(* Logix 5000 project; controller fun_probably 1769-L16ER-BB1B rev 34.12; software revision 34.01 *)

TASK MainTask (continuous, watchdog 500 ms) : MainProgram

MODULES
   Local : 1769-L16ER-BB1B (PointIO 0, rev 34.12)
      Discrete_IO : Embedded (PointIO 1, rev 34.11, Output RPI 20 ms)
           Local:1:I.Data.3   // Main or Troubleshooting Switch
END_MODULES

VAR_GLOBAL   (* controller tags *)
   bestScore : DINT;
   birdDownHit : REAL;
   birdFrontHit : REAL[2];
   birdUpHit : REAL;
   birdXPos : DINT;
   birdYPos : REAL;
   clock : TIMER := (PRE := 50);
   downSpeed : DINT;
   dX : DINT;
   dY : REAL;
   fallFunctionX : COUNTER := (PRE := 10);
   fastestFall : BOOL;
   getOffset1 : BOOL;
   getOffset2 : BOOL;
   GodMode : BOOL;
   gravity : REAL;
   halt : BOOL;
   HMI_Start : BOOL;
   increment : DINT;
   intermediateVal : REAL;
   invertUpSpeed : DINT;
   limit : DINT;
   loseBit : BOOL;
   multiplier : DINT;
   offset : DINT;
   ons1 : BOOL;
   ons10 : BOOL;
   ons11 : BOOL;
   ons12 : BOOL;
   ons13 : BOOL;
   ons14 : BOOL;
   ons15 : BOOL;
   ons16 : BOOL;
   ons2 : BOOL;
   ons3 : BOOL;
   ons4 : BOOL;
   ons5 : BOOL;
   ons6 : BOOL;
   ons7 : BOOL;
   ons8 : BOOL;
   ons9 : BOOL;
   pipe1_collision : BOOL;
   pipe1_reset : BOOL;
   pipe1XPos : DINT;
   pipe1Y : REAL;
   pipe1Ybot : REAL;
   pipe1Yhit : DINT;
   pipe2_collision : BOOL;
   pipe2_reset : BOOL;
   pipe2XPos : DINT;
   pipe2Y : DINT;
   pipe2Ybot : DINT;
   pipe2Yhit : DINT;
   run_pipe2 : BOOL;
   score : COUNTER;
   seed : DINT;
   speed : DINT;
   startCR : BOOL;
   temp_offset : DINT;
   temp_seed : DINT;
   test : REAL[32];
   upSpeed : DINT;
END_VAR

PROGRAM MainProgram   (* main routine MainRoutine *)

ROUTINE MainRoutine   (* ladder *)
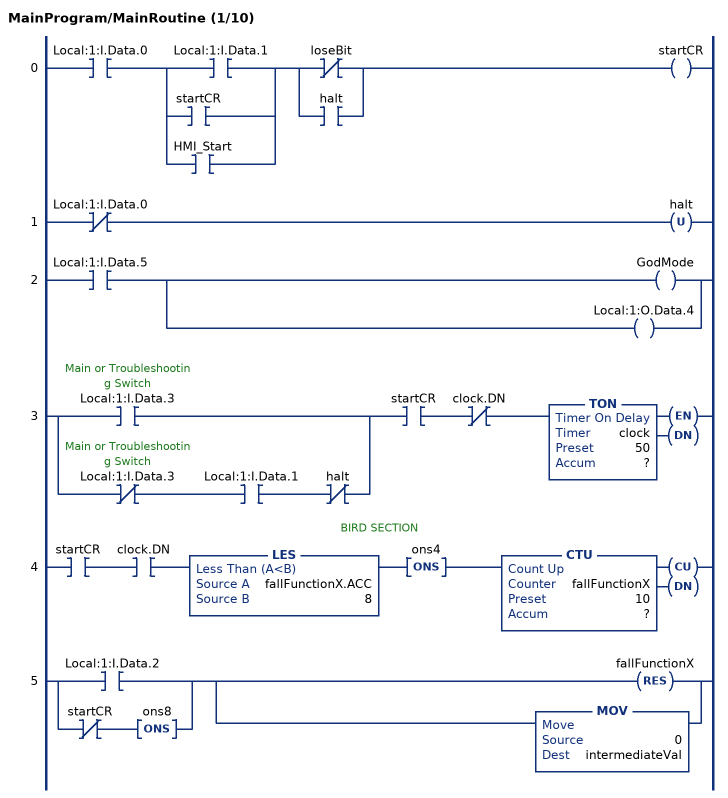
   0: XIC(Local:1:I.Data.0)[XIC(Local:1:I.Data.1) ,[XIC(startCR) ,XIC(HMI_Start) ] ][XIO(loseBit) ,XIC(halt) ]OTE(startCR);
   1: XIO(Local:1:I.Data.0)OTU(halt);
   2: XIC(Local:1:I.Data.5)[OTE(GodMode) ,OTE(Local:1:O.Data.4) ];
   3: [XIC(Local:1:I.Data.3) ,XIO(Local:1:I.Data.3) XIC(Local:1:I.Data.1) XIO(halt) ]XIC(startCR)XIO(clock.DN)TON(clock,?,?);
   // BIRD SECTION
   4: XIC(startCR)XIC(clock.DN)LES(fallFunctionX.ACC,8)ONS(ons4)CTU(fallFunctionX,?,?);
   5: [XIC(Local:1:I.Data.2) ,XIO(startCR) ONS(ons8) ][RES(fallFunctionX) ,MOV(0,intermediateVal) ];
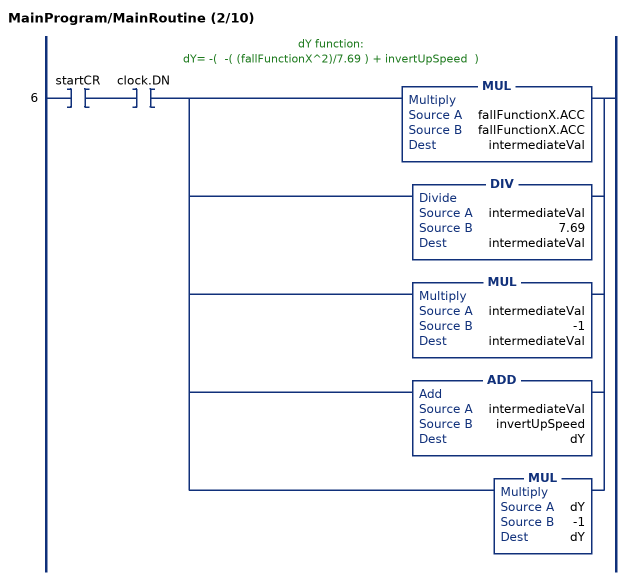
   // dY function:
   // dY= -(  -( (fallFunctionX^2)/7.69 ) + invertUpSpeed  )
   6: XIC(startCR)XIC(clock.DN)[MUL(fallFunctionX.ACC,fallFunctionX.ACC,intermediateVal) ,[DIV(intermediateVal,7.69,intermediateVal) ,[MUL(intermediateVal,-1,intermediateVal) ,[ADD(intermediateVal,invertUpSpeed,dY) ,MUL(dY,-1,dY) ] ] ] ];
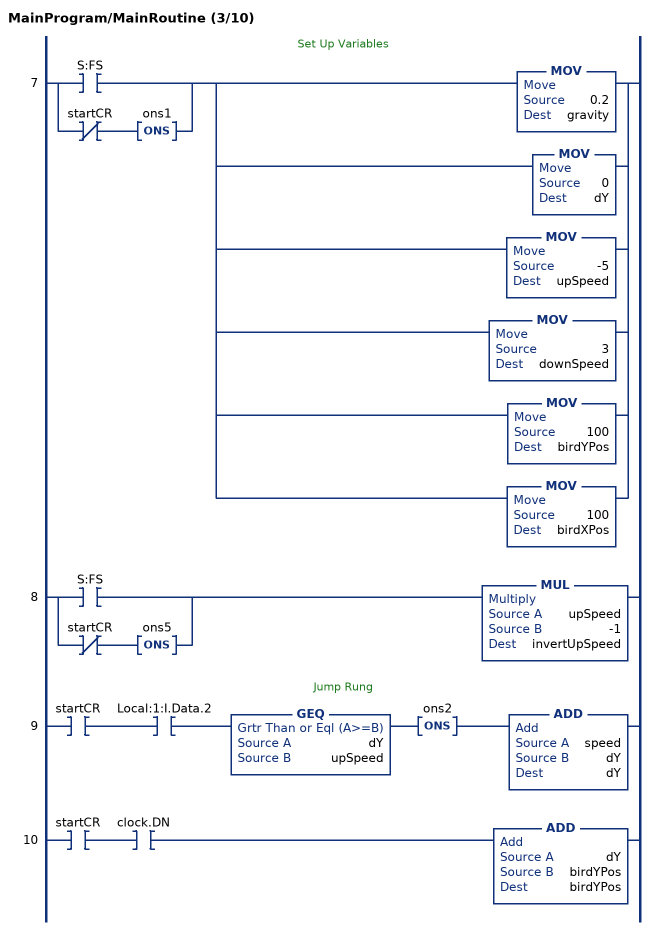
   // Set Up Variables
   7: [XIC(S:FS) ,XIO(startCR) ONS(ons1) ][MOV(0.2,gravity) ,[MOV(0,dY) ,[MOV(-5,upSpeed) ,[MOV(3,downSpeed) ,[MOV(100,birdYPos) ,MOV(100,birdXPos) ] ] ] ] ];
   8: [XIC(S:FS) ,XIO(startCR) ONS(ons5) ]MUL(upSpeed,-1,invertUpSpeed);
   // Jump Rung
   9: XIC(startCR)XIC(Local:1:I.Data.2)GEQ(dY,upSpeed)ONS(ons2)ADD(speed,dY,dY);
   10: XIC(startCR)XIC(clock.DN)ADD(dY,birdYPos,birdYPos);
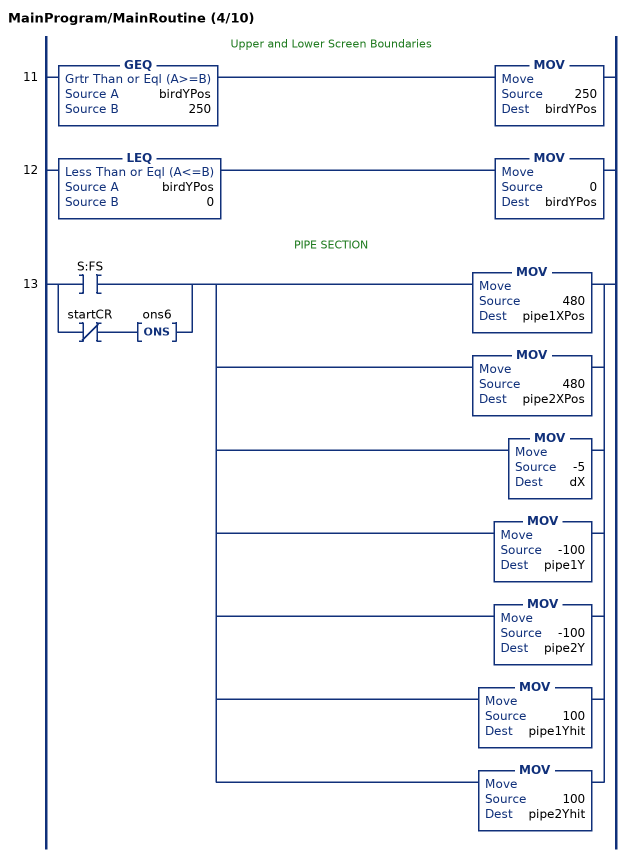
   // Upper and Lower Screen Boundaries
   11: GEQ(birdYPos,250)MOV(250,birdYPos);
   12: LEQ(birdYPos,0)MOV(0,birdYPos);
   // PIPE SECTION
   13: [XIC(S:FS) ,XIO(startCR) ONS(ons6) ][[MOV(480,pipe1XPos) ,MOV(480,pipe2XPos) ] ,[MOV(-5,dX) ,[[MOV(-100,pipe1Y) ,MOV(-100,pipe2Y) ] ,[MOV(100,pipe1Yhit) ,MOV(100,pipe2Yhit) ] ] ] ];
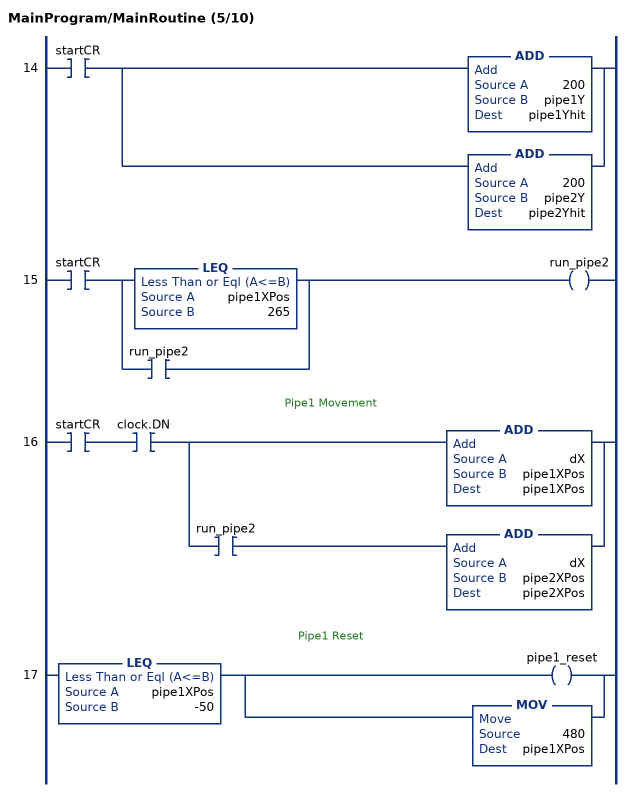
   14: XIC(startCR)[ADD(200,pipe1Y,pipe1Yhit) ,ADD(200,pipe2Y,pipe2Yhit) ];
   15: XIC(startCR)[LEQ(pipe1XPos,265) ,XIC(run_pipe2) ]OTE(run_pipe2);
   // Pipe1 Movement
   16: XIC(startCR)XIC(clock.DN)[ADD(dX,pipe1XPos,pipe1XPos) ,XIC(run_pipe2) ADD(dX,pipe2XPos,pipe2XPos) ];
   // Pipe1 Reset
   17: LEQ(pipe1XPos,-50)[OTE(pipe1_reset) ,MOV(480,pipe1XPos) ];
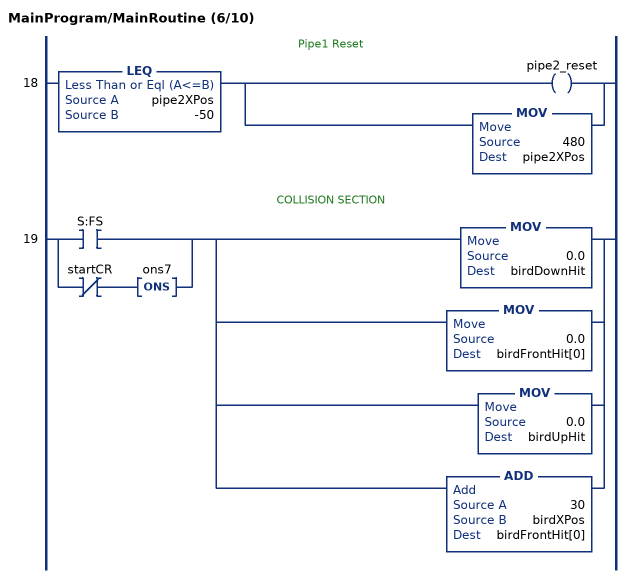
   // Pipe1 Reset
   18: LEQ(pipe2XPos,-50)[OTE(pipe2_reset) ,MOV(480,pipe2XPos) ];
   // COLLISION SECTION
   19: [XIC(S:FS) ,XIO(startCR) ONS(ons7) ][MOV(0.0,birdDownHit) ,[MOV(0.0,birdFrontHit[0]) ,[MOV(0.0,birdUpHit) ,ADD(30,birdXPos,birdFrontHit[0]) ] ] ];
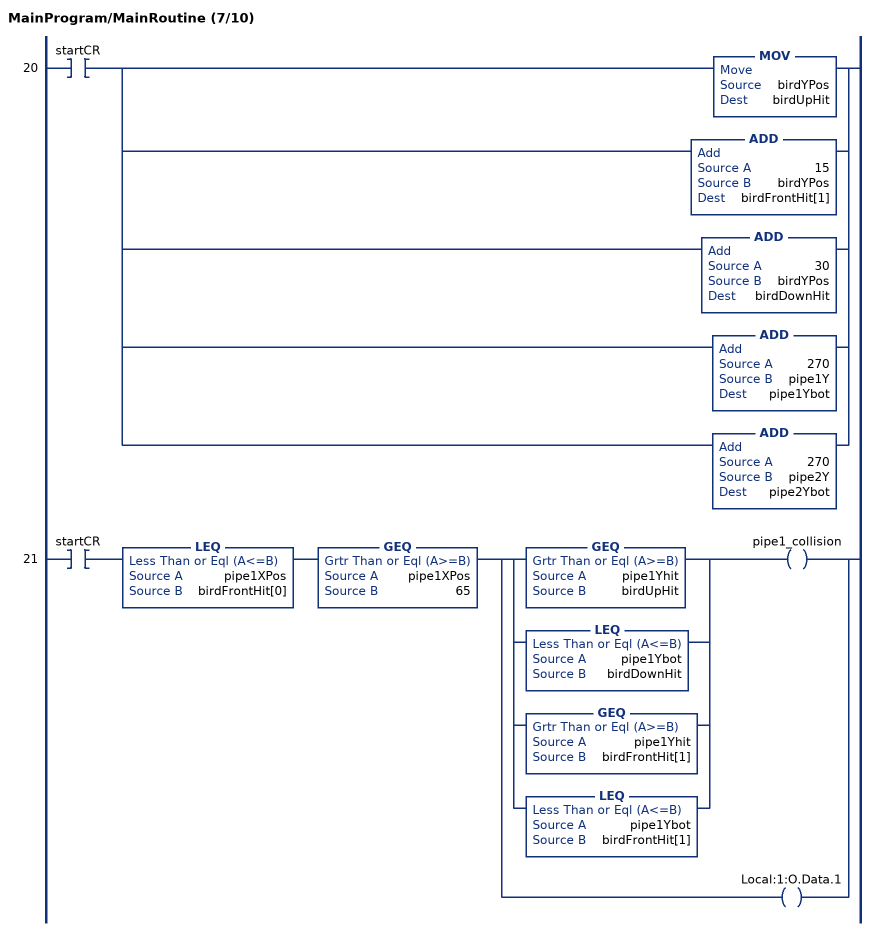
   20: XIC(startCR)[MOV(birdYPos,birdUpHit) ,[ADD(15,birdYPos,birdFrontHit[1]) ,[ADD(30,birdYPos,birdDownHit) ,[ADD(270,pipe1Y,pipe1Ybot) ,ADD(270,pipe2Y,pipe2Ybot) ] ] ] ];
   21: XIC(startCR)LEQ(pipe1XPos,birdFrontHit[0])GEQ(pipe1XPos,65)[[[GEQ(pipe1Yhit,birdUpHit) ,LEQ(pipe1Ybot,birdDownHit) ] ,[GEQ(pipe1Yhit,birdFrontHit[1]) ,LEQ(pipe1Ybot,birdFrontHit[1]) ] ] OTE(pipe1_collision) ,OTE(Local:1:O.Data.1) ];
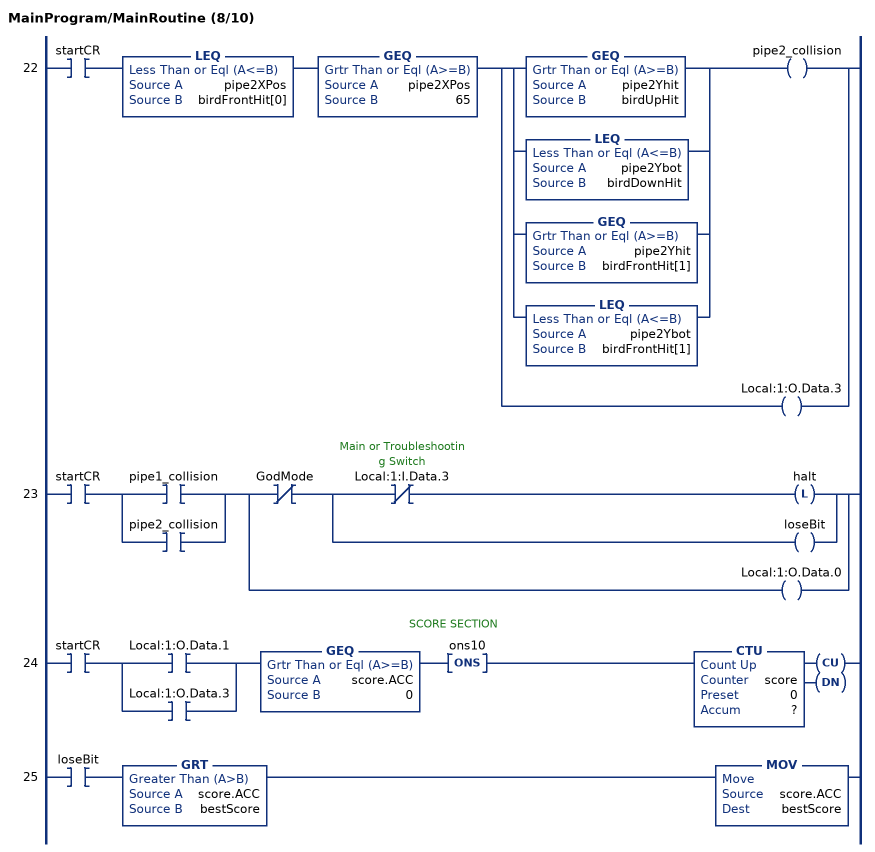
   22: XIC(startCR)LEQ(pipe2XPos,birdFrontHit[0])GEQ(pipe2XPos,65)[[[GEQ(pipe2Yhit,birdUpHit) ,LEQ(pipe2Ybot,birdDownHit) ] ,[GEQ(pipe2Yhit,birdFrontHit[1]) ,LEQ(pipe2Ybot,birdFrontHit[1]) ] ] OTE(pipe2_collision) ,OTE(Local:1:O.Data.3) ];
   23: XIC(startCR)[XIC(pipe1_collision) ,XIC(pipe2_collision) ][XIO(GodMode) [XIO(Local:1:I.Data.3) OTL(halt) ,OTE(loseBit) ] ,OTE(Local:1:O.Data.0) ];
   // SCORE SECTION
   24: XIC(startCR)[XIC(Local:1:O.Data.1) ,XIC(Local:1:O.Data.3) ]GEQ(score.ACC,0)ONS(ons10)CTU(score,?,?);
   25: XIC(loseBit)GRT(score.ACC,bestScore)MOV(score.ACC,bestScore);
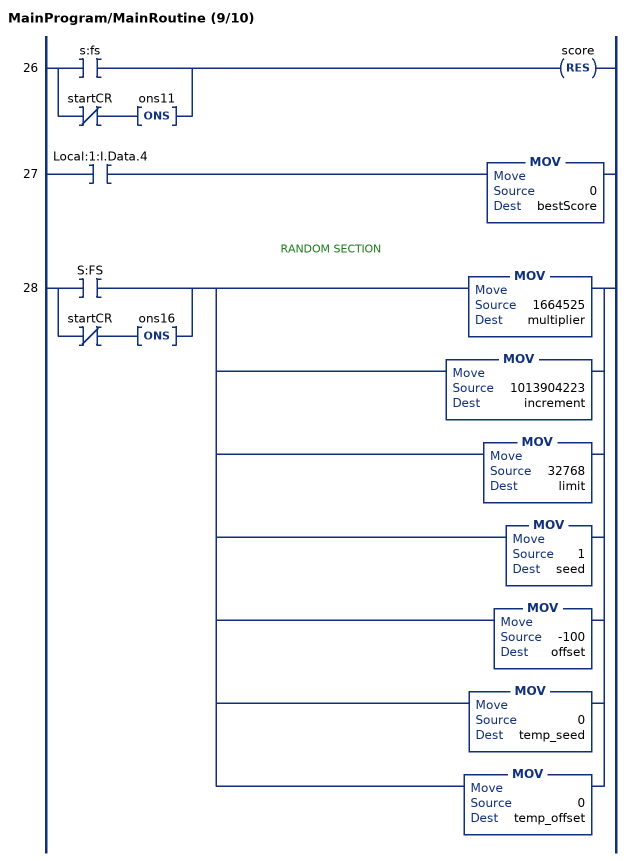
   26: [XIC(s:fs) ,XIO(startCR) ONS(ons11) ]RES(score);
   27: XIC(Local:1:I.Data.4)MOV(0,bestScore);
   // RANDOM SECTION
   28: [XIC(S:FS) ,XIO(startCR) ONS(ons16) ][MOV(1664525,multiplier) ,[MOV(1013904223,increment) ,[MOV(32768,limit) ,[MOV(1,seed) ,[MOV(-100,offset) ,[MOV(0,temp_seed) ,MOV(0,temp_offset) ] ] ] ] ] ];
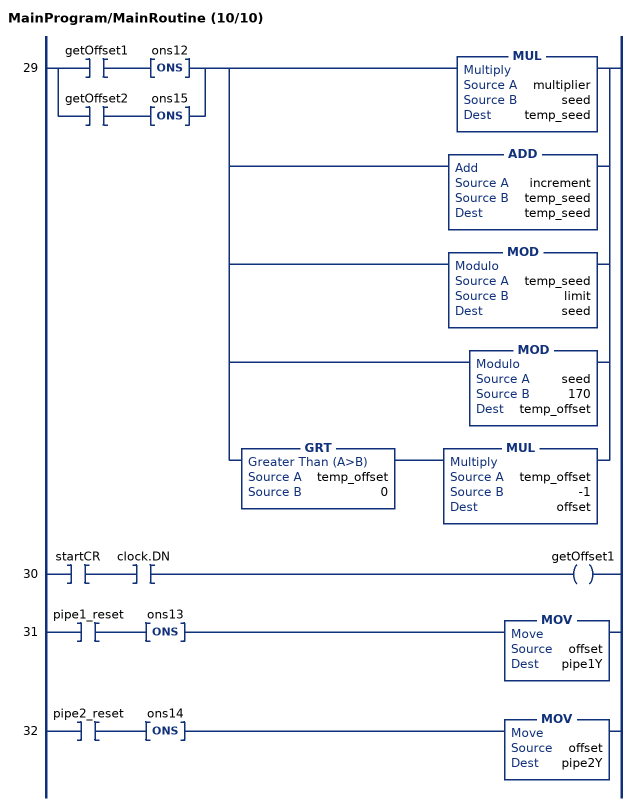
   29: [XIC(getOffset1) ONS(ons12) ,XIC(getOffset2) ONS(ons15) ][MUL(multiplier,seed,temp_seed) ,[ADD(increment,temp_seed,temp_seed) ,[MOD(temp_seed,limit,seed) ,[MOD(seed,170,temp_offset) ,GRT(temp_offset,0) MUL(temp_offset,-1,offset) ] ] ] ];
   30: XIC(startCR)XIC(clock.DN)OTE(getOffset1);
   31: XIC(pipe1_reset)ONS(ons13)MOV(offset,pipe1Y);
   32: XIC(pipe2_reset)ONS(ons14)MOV(offset,pipe2Y);
END_ROUTINE
END_PROGRAM
